VISUALIZATION FouceAutomotiveVisualisation  // 2x2
END_VISUALIZATION

(* stored: Version 1.1.0.1, ProductVersion 3.1.4024.12
   Visu FouceAutomotiveVisualisation: Id {8e228bda-5dc8-4037-8117-89cf82bb03d5} *)
